// TIA Portal V19 export
DATA_BLOCK "MES_Com_Channel_Topic2XX"   // DB29
// stored: Access Published, MemoryReserve 100
   VAR
      RECEIVE : Struct   // Ricezione singolo messaggio da MES
         ack : DInt;   // Acknowledge msg.ID to MES
         msg : "MES_Msg";
      END_STRUCT;
      SEND : Struct   // Invio singolo messaggio a MES
         ack : DInt;   // Acknowledge msg.ID From MES
         msg : "MES_Msg";
      END_STRUCT;
   END_VAR
BEGIN
END_DATA_BLOCK
